(* PLC project capteur_tor, TNI-Software ControlBuild 4.00 *)
(* stored: creationDateTime 2018-09-17T17:24:47-01:00 *)

FUNCTION_BLOCK tapis_conv.capteur_tor
  VAR_INPUT  (* CB.kind=inputVars *)
    Position_IN : REAL := 0.0;
    Position_Fixe : REAL := 0.0;
  END_VAR
  VAR_OUTPUT  (* CB.kind=outputVars *)
    Etat : BOOL := false;
  END_VAR
  VAR CONSTANT  (* CB.kind=parameterVars *)
    Fourchette : REAL := 0.1;
  END_VAR

if Position_IN>(Position_Fixe-Fourchette) and Position_IN<(Position_Fixe+Fourchette)
then
	Etat:=true;
else 
	Etat:=false;
end_if;
END_FUNCTION_BLOCK
